{attribute 'GeneratedUsingTerminal: EL3403-0000-0018'}
{attribute addProperty BoxType "EL3403-0000-0018"}
{attribute addProperty Id "Sync_ErrorAT %I*BOOL1TxPDO_ToggleAT %I*BOOL1CurrentAT %I*DINT4VoltageAT %I*DINT4Active_powerAT %I*DINT4IndexAT %I*USINT1Variant_valueAT %I*DINT4"}
{attribute addProperty CRC "610844445"}
{attribute addProperty Size "19"}
TYPE PM_Inputs_Channel_2468BF1D EXTENDS InputBase_8311D824 :
STRUCT
	{attribute addProperty Name "Sync_Error"}
	Sync_Error AT %I* : BOOL;
	{attribute addProperty Name "TxPDO_Toggle"}
	TxPDO_Toggle AT %I* : BOOL;
	{attribute addProperty Name "Current"}
	Current AT %I* : DINT;
	{attribute addProperty Name "Voltage"}
	Voltage AT %I* : DINT;
	{attribute addProperty Name "Active_power"}
	Active_power AT %I* : DINT;
	{attribute addProperty Name "Index"}
	Index AT %I* : USINT;
	{attribute addProperty Name "Variant_value"}
	Variant_value AT %I* : DINT;
END_STRUCT
END_TYPE

(* stored: Version 1.2.0.0, ProductVersion 3.1.4024.11
   DUT PM_Inputs_Channel_2468BF1D: Id {f0ac9fcb-7a81-4aeb-aae7-61688b76148b} *)
